(* Schneider Machine Expert - Basic project MES_I40_MAC15, file version 2.9.0.0 *)
(* CompanyInformations: Name=BAZZICA *)
(* ProjectInformations: Name=I40BAZZICA, Description=MAC18
PS2075
P00401
IP:192.168.0.161 *)
(* UserInformations: LastName=Dominici, FirstName=Erica, PhoneNumber=+39 0742 38501, Email=info@promas.com, Street=via XXV Aprile, 10/12, City=Trevi, ZipCode=06039, State=Perugia, Country=Italy *)

HARDWARE
  Cpu 0: TM221CE16T
  Cartridge1 0: TMC2TI2
  EthernetConfiguration: NetworkName=M221, IpAllocationMode=FixedAddress, IpAddress=192.168.0.174, SubnetMask=255.255.254.0
  EthernetConfiguration: NetworkName=M221, IpAllocationMode=FixedAddress, IpAddress=0.0.0.0, SubnetMask=0.0.0.0
  SerialLineConfiguration: Baud=Baud19200, Parity=ParityEven, DataBits=DataBits8, StopBits=StopBits1, PhysicalMedium=PhysicalMediumRs485, TransmissionMode=TransmissionModeModbusRtu, SlaveId=1, Addressing=SlaveAddressing
  MastTask: UsePeriodScanMode=true, PeriodScan=100
  FastTask: Period=255
  CpuBehavior: StartingMode=StartAutoRunForced, AutoSaveRamOnEeprom=true, WatchdogPeriod=250

SYMBOLS  (address, symbol, comment, settings)
  %M0       NEW_CYCLE_TRIGGER_V
  %M1       COMMIT_DONE  "COMMIT COMPLETE ACCORDING TO MES/ERP INFO"
  %M40      RUN_S  "RUN"
  %M41      ALARM_S  "ALARM"
  %M42      MOLD_CHG_S  "MOLD CHANGE"
  %M43      MAN_AUT_S  "MAN(1) AUTO(0)"
  %M44      NEW_CYCLE_TRIG_S  "NEW CYCLE TRIGGER"
  %M45      COMMIT_END_S  "COMMIT END"
  %M46      SPARE_1_S  "SPARE 1 S"
  %M400     ONS_1SEC  "ONE SECOND IS ELAPSED"
  %M401     CLOSE_ORDER
  %M402     ONS_1SEC_T
  %S6       SB_TB1S  "Time base of 1 s generated by an internal clock"
  %MW0        "LIFECYCLE COUNTER 1st WORD"
  %MW1      CYCLES_CNT_W1  "LIFECYCEL COUNTER 2nd WORD"
  %MW6      HMI_IN  "HMI_IN"
  %MW7      HMI_OUT  "DATA >> HMI"
  %MW8      HMI_ACTUAL_CYCLE_TIME  "ACTUAL CYCLE TIME"
  %MW9      HMI_LAST_CYCLE_TIME  "LAST CYCLE TIME"
  %MW10     HMI_CYCLES_PER_HOUR  "CYCLES PER HOUR"
  %MW100    ACTUAL_CYCLE_TIME
  %MW101    LAST_CYCLE_TIME
  %MW102    CYCLES_PER_HOURS
  %MD0      CYCLES_CNT_W0
  %TM0      NEW_CYCLE_TRIGGER  [Preset=2, Base=OneSecond]
  %TM1      ONS_1S  [Preset=10, Base=OneHundredMilliSeconds]
  %C0       LIFE_CYCLE_00  "CYCLE COUNTER"  [Preset=0]
  %C1       LIFE_CYCLE_01
  %I0.0     RUN  "MAC GENERAL RELAY ON"
  %I0.1     ALARM  "ALARM"
  %I0.2     MOLD_CHG  "MOLD CHANGE"
  %I0.3     MAN_AUTO  "MACHINE MODE MAN/AUT[1/0]"
  %I0.4     NEW_CYCLE  "NEW CYCLE TRIGGER (AT LOADING)"
  %I0.5     COMMIT_END  "MACHINE REACHED COMMIT TARGET"
  %I0.6       "SPARE"
  %I0.7       "SPARE"
  %I0.8       "SPARE"
  %Q0.0     REMOTE_STOP  "REMOTE STOP"
  %Q0.1     REMOTE_LOAD  "REMOTE RECIPE LOAD CMD"
  %Q0.2     SPARE_02
  %Q0.3     SPARE_03
  %Q0.4     SPARE_04
  %Q0.5     SPARE_05
  %Q0.6     SPARE_06
  %IW0.0      "M_PRESSURE"  [Type=Type_0_10V, Scope=Scope_Normal, Minimum=0, Maximum=1000]
  %IW0.1      "F_PRESSURE"  [Type=Type_0_10V, Scope=Scope_Normal, Minimum=0, Maximum=1000]
  %IW0.100    "M_TEMPERATURE"  [Type=Type_ThermocoupleK, Scope=Scope_Celsius, Minimum=-2000, Maximum=13000]
  %IW0.101    "F_TEMPERATURE"  [Type=Type_ThermocoupleK, Scope=Scope_Celsius, Minimum=-2000, Maximum=13000]

POU IN
  (* SectionNumber=1 *)

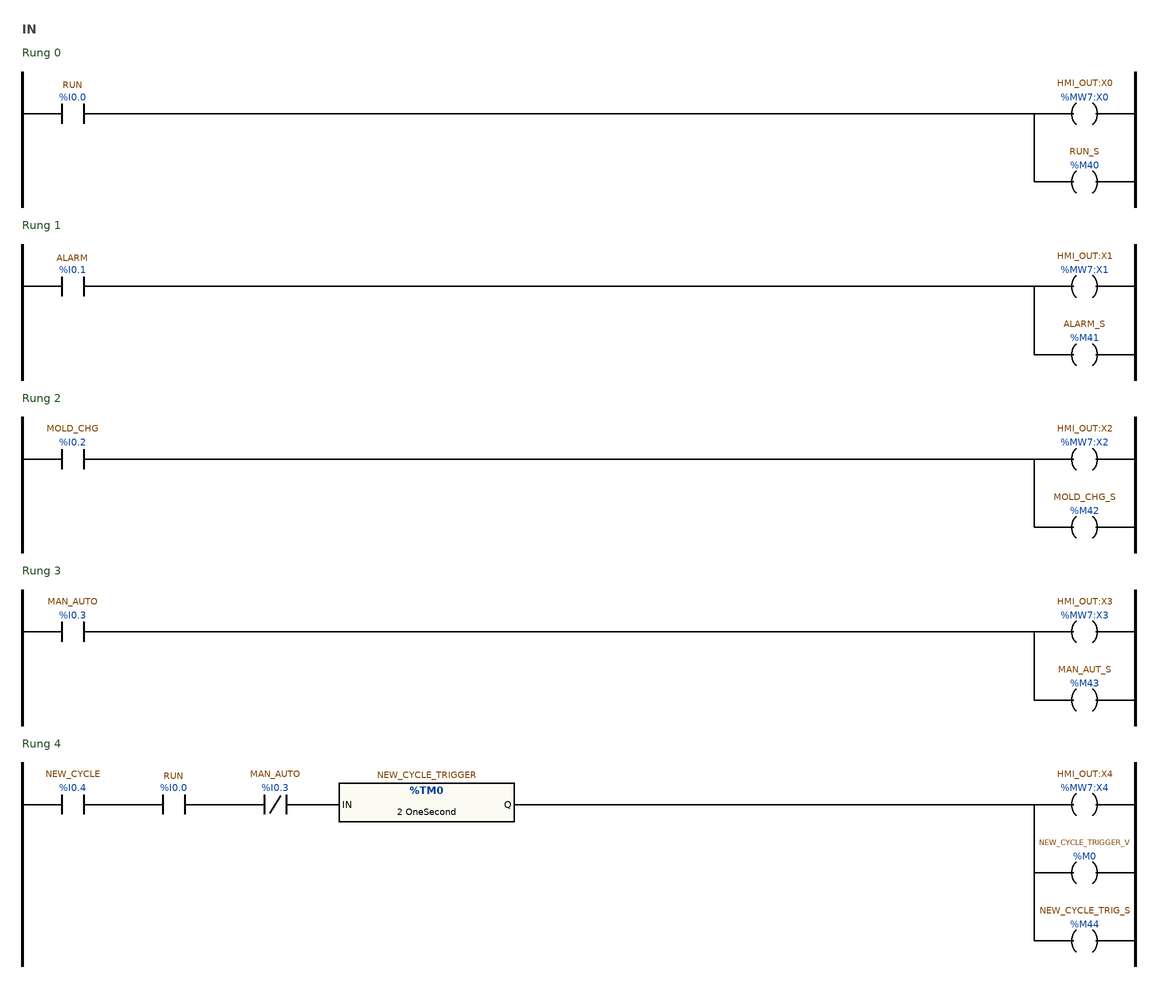

// Rung 0
  LD %I0.0                (* RUN *)
  ST %MW7:X0              (* HMI_OUT *)
  ST %M40                 (* RUN_S *)
  // as ST:
  //   HMI_OUT:X0 := RUN;
  //   RUN_S := RUN;

// Rung 1
  LD %I0.1                (* ALARM *)
  ST %MW7:X1              (* HMI_OUT *)
  ST %M41                 (* ALARM_S *)
  // as ST:
  //   HMI_OUT:X1 := ALARM;
  //   ALARM_S := ALARM;

// Rung 2
  LD %I0.2                (* MOLD_CHG *)
  ST %MW7:X2              (* HMI_OUT *)
  ST %M42                 (* MOLD_CHG_S *)
  // as ST:
  //   HMI_OUT:X2 := MOLD_CHG;
  //   MOLD_CHG_S := MOLD_CHG;

// Rung 3
  LD %I0.3                (* MAN_AUTO *)
  ST %MW7:X3              (* HMI_OUT *)
  ST %M43                 (* MAN_AUT_S *)
  // as ST:
  //   HMI_OUT:X3 := MAN_AUTO;
  //   MAN_AUT_S := MAN_AUTO;

// Rung 4
  BLK %TM0                (* NEW_CYCLE_TRIGGER *)
  LD %I0.4                (* NEW_CYCLE *)
  AND %I0.0               (* RUN *)
  ANDN %I0.3              (* MAN_AUTO *)
  IN
  OUT_BLK
  LD Q
  ST %MW7:X4              (* HMI_OUT *)
  ST %M0                  (* NEW_CYCLE_TRIGGER_V *)
  ST %M44                 (* NEW_CYCLE_TRIG_S *)
  END_BLK
  // as ST:
  //   NEW_CYCLE_TRIGGER(IN := NEW_CYCLE AND RUN AND NOT MAN_AUTO);
  //   HMI_OUT:X4 := NEW_CYCLE_TRIGGER.Q;
  //   NEW_CYCLE_TRIGGER_V := NEW_CYCLE_TRIGGER.Q;
  //   NEW_CYCLE_TRIG_S := NEW_CYCLE_TRIGGER.Q;

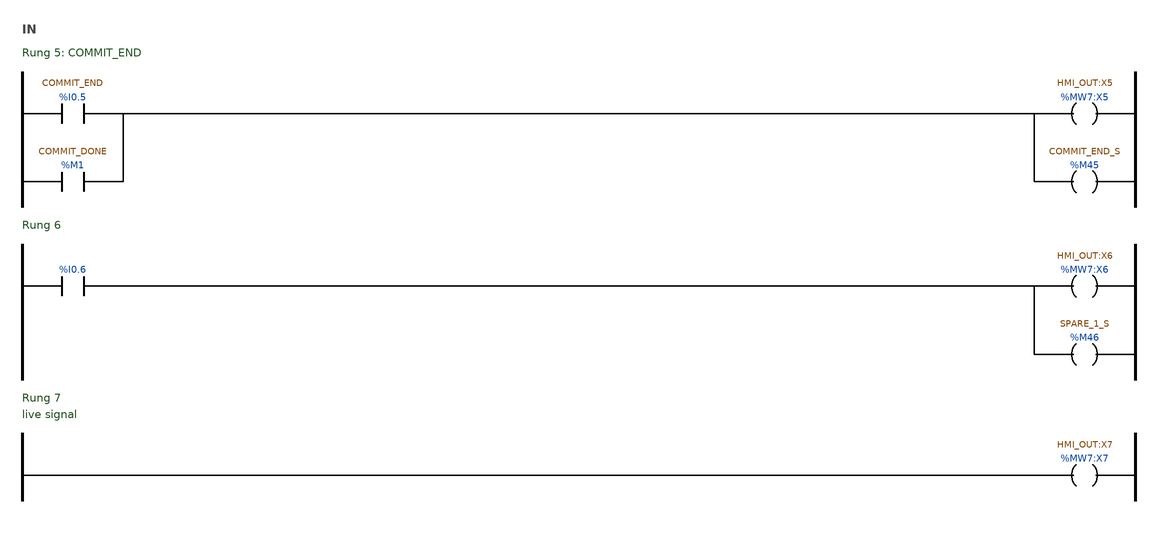

// Rung 5: COMMIT_END
  LD %I0.5                (* COMMIT_END *)
  OR %M1                  (* COMMIT_DONE *)
  ST %MW7:X5              (* HMI_OUT *)
  ST %M45                 (* COMMIT_END_S *)
  // as ST:
  //   HMI_OUT:X5 := COMMIT_END OR COMMIT_DONE;
  //   COMMIT_END_S := COMMIT_END OR COMMIT_DONE;

// Rung 6
  LD %I0.6
  ST %MW7:X6              (* HMI_OUT *)
  ST %M46                 (* SPARE_1_S *)
  // as ST:
  //   HMI_OUT:X6 := %I0.6;
  //   SPARE_1_S := %I0.6;

// Rung 7
// live signal
  LD 1
  ST %MW7:X7              (* HMI_OUT *)
  // as ST:
  //   HMI_OUT:X7 := TRUE;

POU TMR_CNT
  (* SectionNumber=2 *)

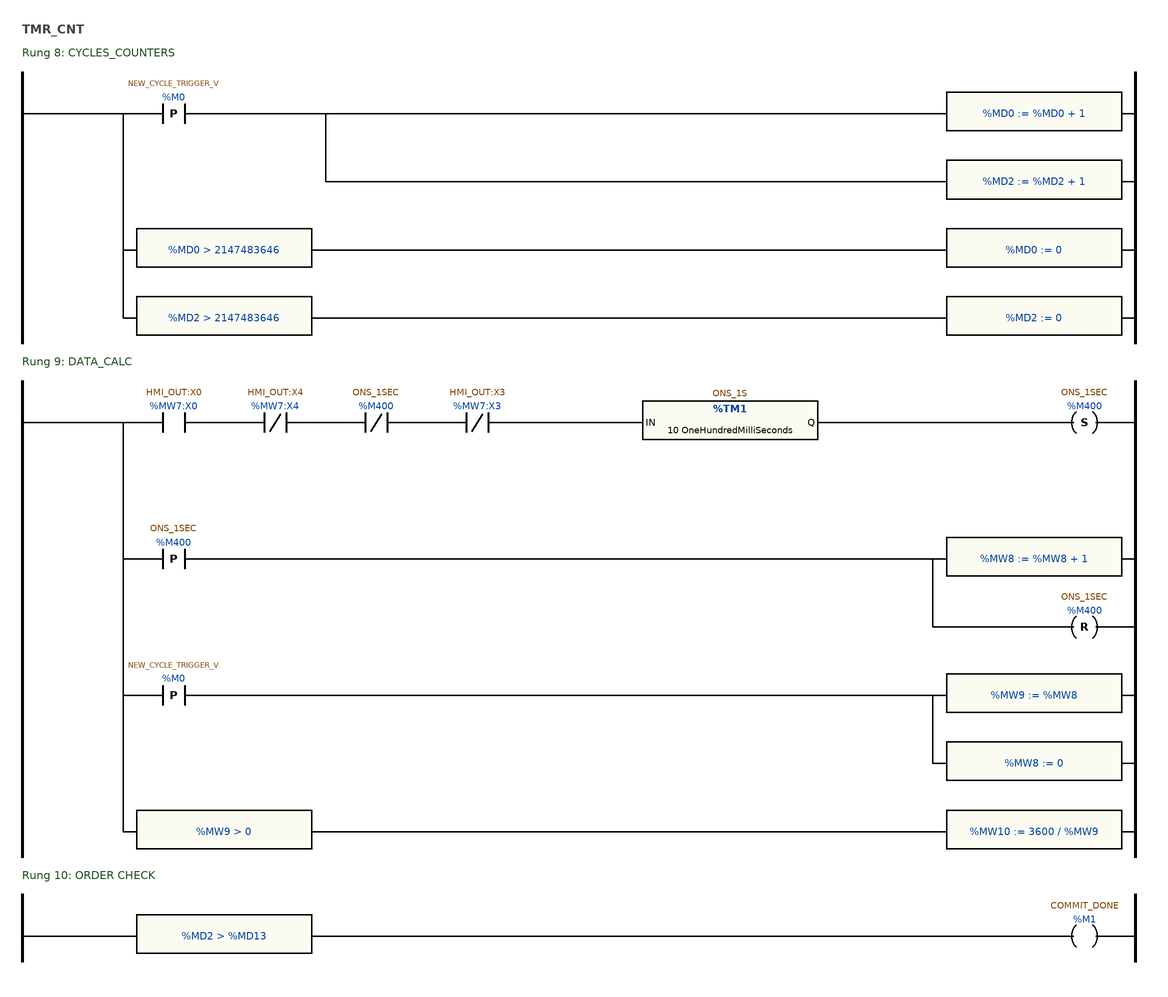

// Rung 8: CYCLES_COUNTERS
  LD 1
  MPS
  ANDR %M0                (* NEW_CYCLE_TRIGGER_V *)
  [ %MD0 := %MD0 + 1 ]    (* CYCLES_CNT_W0, CYCLES_CNT_W0 *)
  [ %MD2 := %MD2 + 1 ]
  MRD
  AND [ %MD0 > 2147483646 ](* CYCLES_CNT_W0 *)
  [ %MD0 := 0 ]           (* CYCLES_CNT_W0 *)
  MPP
  AND [ %MD2 > 2147483646 ]
  [ %MD2 := 0 ]
  // as ST:
  //   IF RISING(NEW_CYCLE_TRIGGER_V) THEN CYCLES_CNT_W0 := CYCLES_CNT_W0 + 1; END_IF;
  //   IF RISING(NEW_CYCLE_TRIGGER_V) THEN %MD2 := %MD2 + 1; END_IF;
  //   IF CYCLES_CNT_W0 > 2147483646 THEN CYCLES_CNT_W0 := 0; END_IF;
  //   IF %MD2 > 2147483646 THEN %MD2 := 0; END_IF;

// Rung 9: DATA_CALC
  LD 1
  MULTIFB
  LD 1
  ST %MW2009:X0
  BLK %TM1                (* ONS_1S *)
  LD %MW2009:X0
  AND %MW7:X0             (* HMI_OUT *)
  ANDN %MW7:X4            (* HMI_OUT *)
  ANDN %M400              (* ONS_1SEC *)
  ANDN %MW7:X3            (* HMI_OUT *)
  IN
  OUT_BLK
  LD Q
  S %M400                 (* ONS_1SEC *)
  END_BLK
  LD %MW2009:X0
  MPS
  ANDR %M400              (* ONS_1SEC *)
  [ %MW8 := %MW8 + 1 ]    (* HMI_ACTUAL_CYCLE_TIME, HMI_ACTUAL_CYCLE_TIME *)
  R %M400                 (* ONS_1SEC *)
  MRD
  ANDR %M0                (* NEW_CYCLE_TRIGGER_V *)
  [ %MW9 := %MW8 ]        (* HMI_LAST_CYCLE_TIME, HMI_ACTUAL_CYCLE_TIME *)
  [ %MW8 := 0 ]           (* HMI_ACTUAL_CYCLE_TIME *)
  MPP
  AND [ %MW9 > 0 ]        (* HMI_LAST_CYCLE_TIME *)
  [ %MW10 := 3600 / %MW9 ](* HMI_CYCLES_PER_HOUR, HMI_LAST_CYCLE_TIME *)
  MULTIFB
  // as ST:
  //   ONS_1S(IN := HMI_OUT:X0 AND NOT HMI_OUT:X4 AND NOT ONS_1SEC AND NOT HMI_OUT:X3);
  //   IF ONS_1S.Q THEN ONS_1SEC := TRUE; END_IF;
  //   IF RISING(ONS_1SEC) THEN HMI_ACTUAL_CYCLE_TIME := HMI_ACTUAL_CYCLE_TIME + 1; END_IF;
  //   IF RISING(ONS_1SEC) THEN ONS_1SEC := FALSE; END_IF;
  //   IF RISING(NEW_CYCLE_TRIGGER_V) THEN HMI_LAST_CYCLE_TIME := HMI_ACTUAL_CYCLE_TIME; END_IF;
  //   IF RISING(NEW_CYCLE_TRIGGER_V) THEN HMI_ACTUAL_CYCLE_TIME := 0; END_IF;
  //   IF HMI_LAST_CYCLE_TIME > 0 THEN HMI_CYCLES_PER_HOUR := 3600 / HMI_LAST_CYCLE_TIME; END_IF;

// Rung 10: ORDER CHECK
  LD 1
  AND [ %MD2 > %MD13 ]
  ST %M1                  (* COMMIT_DONE *)
  // as ST:
  //   COMMIT_DONE := %MD2 > %MD13;

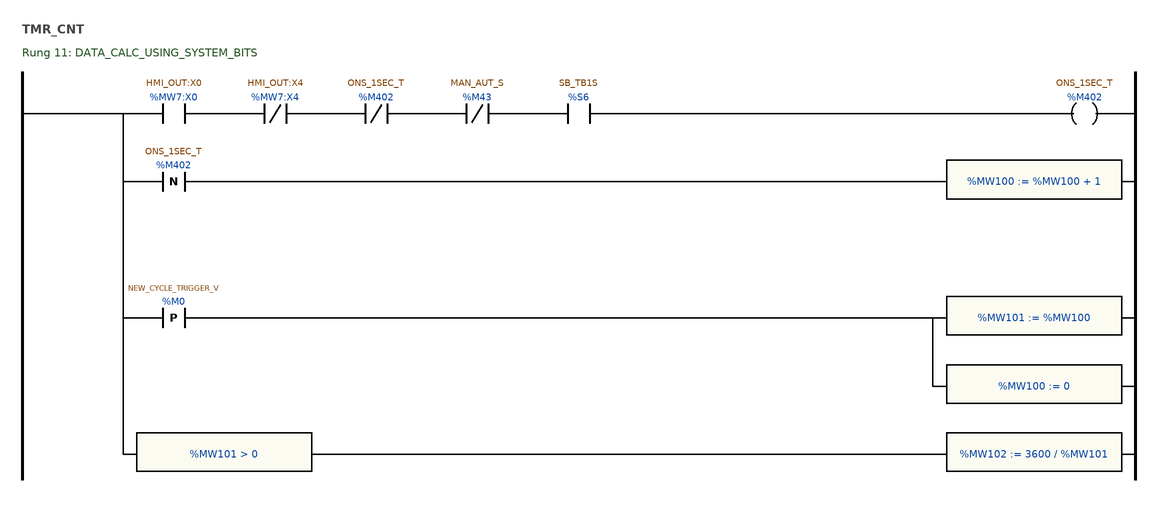

// Rung 11: DATA_CALC_USING_SYSTEM_BITS
  LD 1
  MPS
  AND %MW7:X0             (* HMI_OUT *)
  ANDN %MW7:X4            (* HMI_OUT *)
  ANDN %M402              (* ONS_1SEC_T *)
  ANDN %M43               (* MAN_AUT_S *)
  AND %S6                 (* SB_TB1S *)
  ST %M402                (* ONS_1SEC_T *)
  MRD
  ANDF %M402              (* ONS_1SEC_T *)
  [ %MW100 := %MW100 + 1 ](* ACTUAL_CYCLE_TIME, ACTUAL_CYCLE_TIME *)
  MRD
  ANDR %M0                (* NEW_CYCLE_TRIGGER_V *)
  [ %MW101 := %MW100 ]    (* LAST_CYCLE_TIME, ACTUAL_CYCLE_TIME *)
  [ %MW100 := 0 ]         (* ACTUAL_CYCLE_TIME *)
  MPP
  AND [ %MW101 > 0 ]      (* LAST_CYCLE_TIME *)
  [ %MW102 := 3600 / %MW101 ](* CYCLES_PER_HOURS, LAST_CYCLE_TIME *)
  // as ST:
  //   ONS_1SEC_T := HMI_OUT:X0 AND NOT HMI_OUT:X4 AND NOT ONS_1SEC_T AND NOT MAN_AUT_S AND SB_TB1S;
  //   IF FALLING(ONS_1SEC_T) THEN ACTUAL_CYCLE_TIME := ACTUAL_CYCLE_TIME + 1; END_IF;
  //   IF RISING(NEW_CYCLE_TRIGGER_V) THEN LAST_CYCLE_TIME := ACTUAL_CYCLE_TIME; END_IF;
  //   IF RISING(NEW_CYCLE_TRIGGER_V) THEN ACTUAL_CYCLE_TIME := 0; END_IF;
  //   IF LAST_CYCLE_TIME > 0 THEN CYCLES_PER_HOURS := 3600 / LAST_CYCLE_TIME; END_IF;

POU OUT
  (* SectionNumber=3 *)

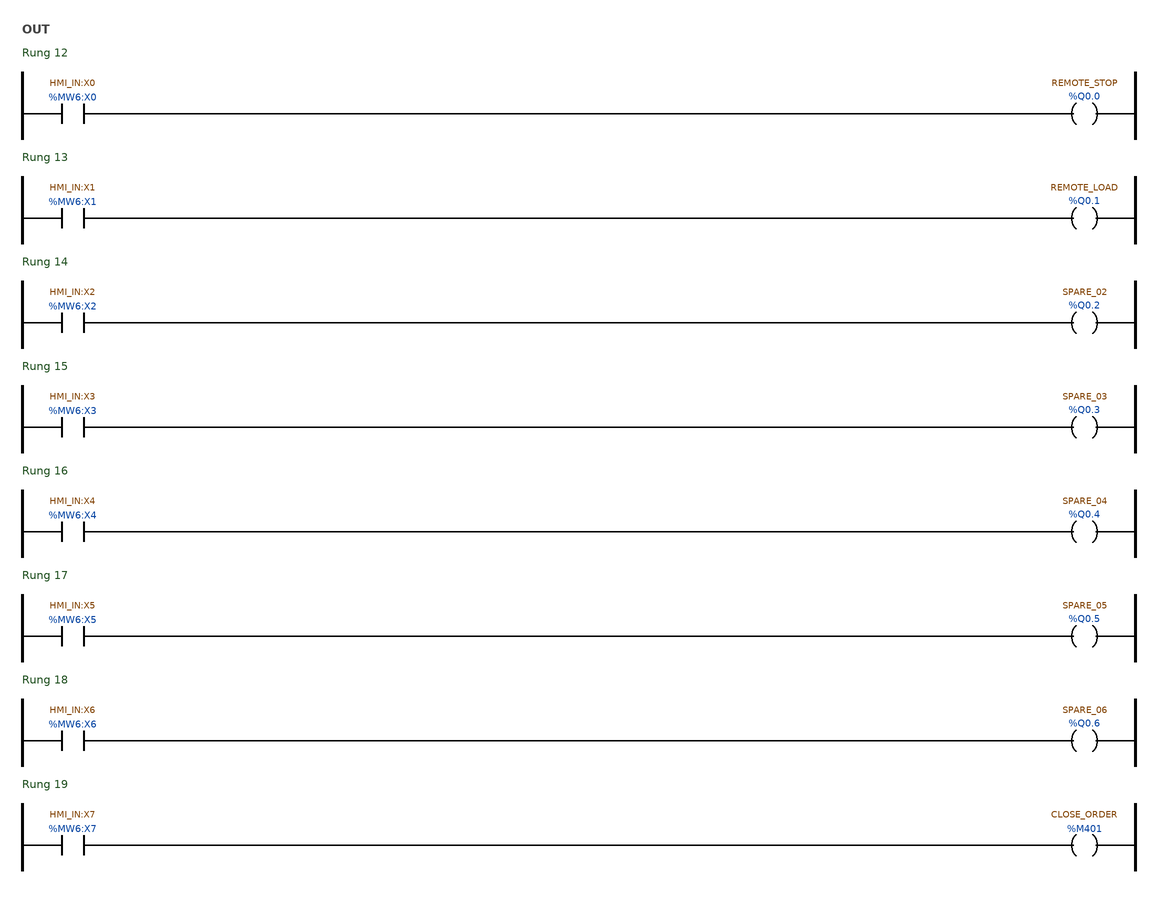

// Rung 12
  LD %MW6:X0              (* HMI_IN *)
  ST %Q0.0                (* REMOTE_STOP *)
  // as ST:
  //   REMOTE_STOP := HMI_IN:X0;

// Rung 13
  LD %MW6:X1              (* HMI_IN *)
  ST %Q0.1                (* REMOTE_LOAD *)
  // as ST:
  //   REMOTE_LOAD := HMI_IN:X1;

// Rung 14
  LD %MW6:X2              (* HMI_IN *)
  ST %Q0.2                (* SPARE_02 *)
  // as ST:
  //   SPARE_02 := HMI_IN:X2;

// Rung 15
  LD %MW6:X3              (* HMI_IN *)
  ST %Q0.3                (* SPARE_03 *)
  // as ST:
  //   SPARE_03 := HMI_IN:X3;

// Rung 16
  LD %MW6:X4              (* HMI_IN *)
  ST %Q0.4                (* SPARE_04 *)
  // as ST:
  //   SPARE_04 := HMI_IN:X4;

// Rung 17
  LD %MW6:X5              (* HMI_IN *)
  ST %Q0.5                (* SPARE_05 *)
  // as ST:
  //   SPARE_05 := HMI_IN:X5;

// Rung 18
  LD %MW6:X6              (* HMI_IN *)
  ST %Q0.6                (* SPARE_06 *)
  // as ST:
  //   SPARE_06 := HMI_IN:X6;

// Rung 19
  LD %MW6:X7              (* HMI_IN *)
  ST %M401                (* CLOSE_ORDER *)
  // as ST:
  //   CLOSE_ORDER := HMI_IN:X7;
